// TIA Portal V16 export
// export: Created 2021-07-03T21:22:43.1063797Z, ExportSetting WithDefaults, DisplayName Totally Integrated Automation Portal, DisplayVersion V16, DisplayName TIA Portal Version Control Interface, DisplayVersion V16, DisplayName TIA Portal Openness, DisplayVersion V16, DisplayName STEP 7 Professional, DisplayVersion V16, DisplayName STEP 7 Safety, DisplayVersion V16, DisplayName WinCC Professional, DisplayVersion V16
TYPE "118MK2_UPIF_Status"
// stored: IsFailsafeCompliant false
   STRUCT
      PLANT_TAG_NAME { ExternalAccessible := 'False'; ExternalVisible := 'False'; ExternalWritable := 'False'} : Array[0..15] of Byte;   // Current plant tag name of the sorting module, 16 character string
      UP_MACHINE_NAME { ExternalAccessible := 'False'; ExternalVisible := 'False'; ExternalWritable := 'False'} : Array[0..15] of Byte;   // Current manufacturer name of the sorting module – read from the cRIO Controller configuration, 16-character string
      COMMAND_ACK_S { ExternalAccessible := 'False'; ExternalVisible := 'False'; ExternalWritable := 'False'} : Byte;   // Returns the (same) command value as an acknowledgement that the Real-time system has received the command.
      COMMAND_IN_PROG_S { ExternalAccessible := 'False'; ExternalVisible := 'False'; ExternalWritable := 'False'} : Byte;   // Counts up as progress indicator – resets on completion
      INVALID_COMMAND_S { ExternalAccessible := 'False'; ExternalVisible := 'False'; ExternalWritable := 'False'} : Bool;   // ‘1’ when an invalid command – cleared on next valid command.
      PARAM_OUT_OF_RANGE_S { ExternalAccessible := 'False'; ExternalVisible := 'False'; ExternalWritable := 'False'} : Bool;   // ‘1’ when any requested parameter value is out of range.
      USER_ADDED_S { ExternalAccessible := 'False'; ExternalVisible := 'False'; ExternalWritable := 'False'} : Bool;   // ‘1’ when a requested new user name was successfully added to the security lookup table.
      PASSWORD_CHANGED_S { ExternalAccessible := 'False'; ExternalVisible := 'False'; ExternalWritable := 'False'} : Bool;   // ‘1’ when a requested password change was successful.
      USER_DELETED_S { ExternalAccessible := 'False'; ExternalVisible := 'False'; ExternalWritable := 'False'} : Bool;   // ‘1’ temporarily when a requested user delete was successful
      LOGON_ATTEMPT_FAILED_S { ExternalAccessible := 'False'; ExternalVisible := 'False'; ExternalWritable := 'False'} : Bool;   // ‘1’ temporarily when a logon attempt failed.
      NO_XRAY_DOOR_OPEN_S { ExternalAccessible := 'False'; ExternalVisible := 'False'; ExternalWritable := 'False'} : Bool;   // ‘1’ temporarily when no X-rays possible because doors are open.
      NO_OPP_INCOM_AIR_LOW_S { ExternalAccessible := 'False'; ExternalVisible := 'False'; ExternalWritable := 'False'} : Bool;   // ‘1’ temporarily when no operation possible due to low air pressure.
      GLOBAL_ALARM_S { ExternalAccessible := 'False'; ExternalVisible := 'False'; ExternalWritable := 'False'} : Bool;   // ‘1’ when any alarm is present. Cleared when all alarms are reset.
      OTI_COMMS_FAULT_S { ExternalAccessible := 'False'; ExternalVisible := 'False'; ExternalWritable := 'False'} : Bool;   // ‘1’ when comms fault between OTI and cRIO.
      LOCAL_REMOTE_S { ExternalAccessible := 'False'; ExternalVisible := 'False'; ExternalWritable := 'False'} : Bool;   // ‘1’ when machine is in Remote mode
      MAINTENANCE_MODE_S { ExternalAccessible := 'False'; ExternalVisible := 'False'; ExternalWritable := 'False'} : Bool;   // ‘1’ when in Maintenance Mode
      INCOM_AIR_PRESS_LO_S { ExternalAccessible := 'False'; ExternalVisible := 'False'; ExternalWritable := 'False'} : Bool;   // ‘1’ when incoming air pressure less than low setpoint i.e. 4.5 bar.
      INCOM_AIR_PRESS_LOLO_S { ExternalAccessible := 'False'; ExternalVisible := 'False'; ExternalWritable := 'False'} : Bool;   // ‘1’ when incoming air pressure less than low low setpoint i.e. 4.0 bar.
      PROC_WATERFLOW_HIGH_S { ExternalAccessible := 'False'; ExternalVisible := 'False'; ExternalWritable := 'False'} : Bool;   // ‘1’ when flow rate greater than flow set-point plus allowed deviation.
      PROC_WATERFLOW_LOW_S { ExternalAccessible := 'False'; ExternalVisible := 'False'; ExternalWritable := 'False'} : Bool;   // ‘1’ when flow rate less than flow set-point minus allowed deviation.
      FEEDER_RUNNING_S { ExternalAccessible := 'False'; ExternalVisible := 'False'; ExternalWritable := 'False'} : Bool;   // ‘1’ when feeder is running.
      REMOTE_DNSTRM_INTLK_S { ExternalAccessible := 'False'; ExternalVisible := 'False'; ExternalWritable := 'False'} : Bool;   // ‘1’ when downstream interlock healthy from PLC.
      HOLD_STATE_S { ExternalAccessible := 'False'; ExternalVisible := 'False'; ExternalWritable := 'False'} : Bool;   // ‘1’ when feeder is prevented from running in “Processing” due to process interlock, low air pressure etc.
      WAIT_STATE_S { ExternalAccessible := 'False'; ExternalVisible := 'False'; ExternalWritable := 'False'} : Bool;   // ‘1’ when in “Processing” state.
      PURGED_STATE_S { ExternalAccessible := 'False'; ExternalVisible := 'False'; ExternalWritable := 'False'} : Bool;   // ‘1’ when a purge cycle is successfully completed. Cleared when feeder is next started.
      EJECTION_RATE_WARN_S { ExternalAccessible := 'False'; ExternalVisible := 'False'; ExternalWritable := 'False'} : Bool;   // ‘1’ when ejection rate exceeds warning level.
      EJECTION_RATE_ALARM_S { ExternalAccessible := 'False'; ExternalVisible := 'False'; ExternalWritable := 'False'} : Bool;   // ‘1’ when ejection rate exceeded ejection rate alarm level.
      MACH_ESTOP_ACTIVE_S { ExternalAccessible := 'False'; ExternalVisible := 'False'; ExternalWritable := 'False'} : Bool;   // ‘1’ when E-stop active.
      XRAY_COOLW_TEMP_FAULT_S { ExternalAccessible := 'False'; ExternalVisible := 'False'; ExternalWritable := 'False'} : Bool;   // ‘1’ when X-ray cooling water temperature to high or too low fault detected.
      XRAY_COOLW_FLOW_FAULT_S { ExternalAccessible := 'False'; ExternalVisible := 'False'; ExternalWritable := 'False'} : Bool;   // ‘1’ when cooling water flow low fault detected.
      PROC_WATER_FLOW_S { ExternalAccessible := 'False'; ExternalVisible := 'False'; ExternalWritable := 'False'} : Bool;   // ‘1’ when process water flow too high or too low fault detected. (Wet machine only)
      FRONT_SIDE_PROC_DOOR_S { ExternalAccessible := 'False'; ExternalVisible := 'False'; ExternalWritable := 'False'} : Bool;   // ‘1’ when front side door open.
      BACK_SIDE_PROC_DOOR_S { ExternalAccessible := 'False'; ExternalVisible := 'False'; ExternalWritable := 'False'} : Bool;   // ‘1’ when back side door open.
      FEEDER_DOOR_S { ExternalAccessible := 'False'; ExternalVisible := 'False'; ExternalWritable := 'False'} : Bool;   // ‘1’ when feeder door open.
      HOOD_S { ExternalAccessible := 'False'; ExternalVisible := 'False'; ExternalWritable := 'False'} : Bool;   // ‘1’ when hood open.
      CONC_TRACER_DOOR_S { ExternalAccessible := 'False'; ExternalVisible := 'False'; ExternalWritable := 'False'} : Bool;   // ‘1’ when concentrate tracer door open.
      TAILINGS_TRACER_DOOR_S { ExternalAccessible := 'False'; ExternalVisible := 'False'; ExternalWritable := 'False'} : Bool;   // ‘1’ when tailings tracer door open.
      CONC_TRACER_TRAY_S { ExternalAccessible := 'False'; ExternalVisible := 'False'; ExternalWritable := 'False'} : Bool;   // ‘1’ when concentrate tracer tray in position.
      TAILINGS_TRACER_TRAY_S { ExternalAccessible := 'False'; ExternalVisible := 'False'; ExternalWritable := 'False'} : Bool;   // ‘1’ when tailings tracer tray in position.
      PLANT_INLET_CHUTE_S { ExternalAccessible := 'False'; ExternalVisible := 'False'; ExternalWritable := 'False'} : Bool;   // ‘1’ when plant inlet not in position.
      INSPECTION_COVER_S { ExternalAccessible := 'False'; ExternalVisible := 'False'; ExternalWritable := 'False'} : Bool;   // ‘1’ when inspection cover not in position.
      PLANT_CONC_CHUTE_S { ExternalAccessible := 'False'; ExternalVisible := 'False'; ExternalWritable := 'False'} : Bool;   // ‘1’ when plant concentrate chute not in position.
      PLANT_TAILINGS_CHUTE_S { ExternalAccessible := 'False'; ExternalVisible := 'False'; ExternalWritable := 'False'} : Bool;   // ‘1’ when plant tailings chute not in position.
      INTERN_CONC_CHUTE_S { ExternalAccessible := 'False'; ExternalVisible := 'False'; ExternalWritable := 'False'} : Bool;   // ‘1’ when internal concentrate chute not in position.
      INTERN_TAILINGS_CHUTE_S { ExternalAccessible := 'False'; ExternalVisible := 'False'; ExternalWritable := 'False'} : Bool;   // ‘1’ when internal tailings chute not in position.
      DUSTEXTRACT_FLOW_FLT_S { ExternalAccessible := 'False'; ExternalVisible := 'False'; ExternalWritable := 'False'} : Bool;   // ‘1’ when dust extractor flow fault detected (Dry machine only)
      SURGE_ARRESTOR_FLT_S { ExternalAccessible := 'False'; ExternalVisible := 'False'; ExternalWritable := 'False'} : Bool;   // ‘1’ when one or more surge arrestors on the electrical panel is faulty.
      DXM_XRAY_GEN_COMM_FLT_S { ExternalAccessible := 'False'; ExternalVisible := 'False'; ExternalWritable := 'False'} : Bool;   // ‘1’ when no comms between cRIO and Spellman DXM X-ray generator.
      DXM_HV_ENABLED_S { ExternalAccessible := 'False'; ExternalVisible := 'False'; ExternalWritable := 'False'} : Bool;   // ‘1’ when X-rays ON.
      DXM_INTERLOCK_CLOSED_S { ExternalAccessible := 'False'; ExternalVisible := 'False'; ExternalWritable := 'False'} : Bool;   // ‘1’ when interlock on X-ray generator is healthy.
      DXM_PS_FLT_S { ExternalAccessible := 'False'; ExternalVisible := 'False'; ExternalWritable := 'False'} : Bool;   // ‘1’ when X-ray generator power supply fault detected.
      STATUS_BYTE6_SPARE7 { ExternalAccessible := 'False'; ExternalVisible := 'False'; ExternalWritable := 'False'} : Bool;   // Status Byte-6 Spare
      STATUS_BYTE7_SPARE0 { ExternalAccessible := 'False'; ExternalVisible := 'False'; ExternalWritable := 'False'} : Bool;   // Status Byte-7 Spare
      STATUS_BYTE7_SPARE1 { ExternalAccessible := 'False'; ExternalVisible := 'False'; ExternalWritable := 'False'} : Bool;   // Status Byte-7 Spare
      STATUS_BYTE7_SPARE2 { ExternalAccessible := 'False'; ExternalVisible := 'False'; ExternalWritable := 'False'} : Bool;   // Status Byte-7 Spare
      STATUS_BYTE7_SPARE3 { ExternalAccessible := 'False'; ExternalVisible := 'False'; ExternalWritable := 'False'} : Bool;   // Status Byte-7 Spare
      STATUS_BYTE7_SPARE4 { ExternalAccessible := 'False'; ExternalVisible := 'False'; ExternalWritable := 'False'} : Bool;   // Status Byte-7 Spare
      STATUS_BYTE7_SPARE5 { ExternalAccessible := 'False'; ExternalVisible := 'False'; ExternalWritable := 'False'} : Bool;   // Status Byte-7 Spare
      STATUS_BYTE7_SPARE6 { ExternalAccessible := 'False'; ExternalVisible := 'False'; ExternalWritable := 'False'} : Bool;   // Status Byte-7 Spare
      STATUS_BYTE7_SPARE7 { ExternalAccessible := 'False'; ExternalVisible := 'False'; ExternalWritable := 'False'} : Bool;   // Status Byte-7 Spare
      STATUS_BYTE8_SPARE0 { ExternalAccessible := 'False'; ExternalVisible := 'False'; ExternalWritable := 'False'} : Bool;   // Status Byte-8 Spare
      STATUS_BYTE8_SPARE1 { ExternalAccessible := 'False'; ExternalVisible := 'False'; ExternalWritable := 'False'} : Bool;   // Status Byte-8 Spare
      STATUS_BYTE8_SPARE2 { ExternalAccessible := 'False'; ExternalVisible := 'False'; ExternalWritable := 'False'} : Bool;   // Status Byte-8 Spare
      STATUS_BYTE8_SPARE3 { ExternalAccessible := 'False'; ExternalVisible := 'False'; ExternalWritable := 'False'} : Bool;   // Status Byte-8 Spare
      STATUS_BYTE8_SPARE4 { ExternalAccessible := 'False'; ExternalVisible := 'False'; ExternalWritable := 'False'} : Bool;   // Status Byte-8 Spare
      STATUS_BYTE8_SPARE5 { ExternalAccessible := 'False'; ExternalVisible := 'False'; ExternalWritable := 'False'} : Bool;   // Status Byte-8 Spare
      STATUS_BYTE8_SPARE6 { ExternalAccessible := 'False'; ExternalVisible := 'False'; ExternalWritable := 'False'} : Bool;   // Status Byte-8 Spare
      STATUS_BYTE8_SPARE7 { ExternalAccessible := 'False'; ExternalVisible := 'False'; ExternalWritable := 'False'} : Bool;   // Status Byte-8 Spare
      STATUS_BYTE9_SPARE0 { ExternalAccessible := 'False'; ExternalVisible := 'False'; ExternalWritable := 'False'} : Bool;   // Status Byte-9 Spare
      STATUS_BYTE9_SPARE1 { ExternalAccessible := 'False'; ExternalVisible := 'False'; ExternalWritable := 'False'} : Bool;   // Status Byte-9 Spare
      STATUS_BYTE9_SPARE2 { ExternalAccessible := 'False'; ExternalVisible := 'False'; ExternalWritable := 'False'} : Bool;   // Status Byte-9 Spare
      STATUS_BYTE9_SPARE3 { ExternalAccessible := 'False'; ExternalVisible := 'False'; ExternalWritable := 'False'} : Bool;   // Status Byte-9 Spare
      STATUS_BYTE9_SPARE4 { ExternalAccessible := 'False'; ExternalVisible := 'False'; ExternalWritable := 'False'} : Bool;   // Status Byte-9 Spare
      STATUS_BYTE9_SPARE5 { ExternalAccessible := 'False'; ExternalVisible := 'False'; ExternalWritable := 'False'} : Bool;   // Status Byte-9 Spare
      STATUS_BYTE9_SPARE6 { ExternalAccessible := 'False'; ExternalVisible := 'False'; ExternalWritable := 'False'} : Bool;   // Status Byte-9 Spare
      STATUS_BYTE9_SPARE7 { ExternalAccessible := 'False'; ExternalVisible := 'False'; ExternalWritable := 'False'} : Bool;   // Status Byte-9 Spare
      STATUS_BYTE10_SPARE0 { ExternalAccessible := 'False'; ExternalVisible := 'False'; ExternalWritable := 'False'} : Bool;   // Status Byte-10 Spare
      STATUS_BYTE10_SPARE1 { ExternalAccessible := 'False'; ExternalVisible := 'False'; ExternalWritable := 'False'} : Bool;   // Status Byte-10 Spare
      STATUS_BYTE10_SPARE2 { ExternalAccessible := 'False'; ExternalVisible := 'False'; ExternalWritable := 'False'} : Bool;   // Status Byte-10 Spare
      STATUS_BYTE10_SPARE3 { ExternalAccessible := 'False'; ExternalVisible := 'False'; ExternalWritable := 'False'} : Bool;   // Status Byte-10 Spare
      STATUS_BYTE10_SPARE4 { ExternalAccessible := 'False'; ExternalVisible := 'False'; ExternalWritable := 'False'} : Bool;   // Status Byte-10 Spare
      STATUS_BYTE10_SPARE5 { ExternalAccessible := 'False'; ExternalVisible := 'False'; ExternalWritable := 'False'} : Bool;   // Status Byte-10 Spare
      STATUS_BYTE10_SPARE6 { ExternalAccessible := 'False'; ExternalVisible := 'False'; ExternalWritable := 'False'} : Bool;   // Status Byte-10 Spare
      STATUS_BYTE10_SPARE7 { ExternalAccessible := 'False'; ExternalVisible := 'False'; ExternalWritable := 'False'} : Bool;   // Status Byte-10 Spare
      MACHINE_STATE_S { ExternalAccessible := 'False'; ExternalVisible := 'False'; ExternalWritable := 'False'} : Byte;   // 0-Initializing, 1-Ready, 2-Purging, 3-Display, 4-Calibrating, 5-Checker Cycle, 6-Processing Ready, 7-Processing, 8-Transition, 9-Alarm.
      DXM_COMMS_FLT_A { ExternalAccessible := 'False'; ExternalVisible := 'False'; ExternalWritable := 'False'} : Bool;   // ALARM: DXM Comms fault
      DXM_XRAY_STATE_A { ExternalAccessible := 'False'; ExternalVisible := 'False'; ExternalWritable := 'False'} : Bool;   // ALARM: DXM X-ray state alarm
      DXM_INTERLOCK_FLT_A { ExternalAccessible := 'False'; ExternalVisible := 'False'; ExternalWritable := 'False'} : Bool;   // ALARM: DXM Interlock fault
      DXM_PSU_FAULT_A { ExternalAccessible := 'False'; ExternalVisible := 'False'; ExternalWritable := 'False'} : Bool;   // ALARM: DXM Power supply fault
      DXM_NOTIN_REM_MODE_A { ExternalAccessible := 'False'; ExternalVisible := 'False'; ExternalWritable := 'False'} : Bool;   // ALARM: DXM Not in remote mode fault
      DXM_ARC_FLT_A { ExternalAccessible := 'False'; ExternalVisible := 'False'; ExternalWritable := 'False'} : Bool;   // ALARM: DXM Arc fault
      DXM_OVER_TEMP_FLT_A { ExternalAccessible := 'False'; ExternalVisible := 'False'; ExternalWritable := 'False'} : Bool;   // ALARM: DXM Over temperature fault
      DXM_OVER_VOLT_FLT_A { ExternalAccessible := 'False'; ExternalVisible := 'False'; ExternalWritable := 'False'} : Bool;   // ALARM: DXM Over voltage fault
      DXM_UNDER_VOLT_FLT_A { ExternalAccessible := 'False'; ExternalVisible := 'False'; ExternalWritable := 'False'} : Bool;   // ALARM: DXM Under voltage fault
      DXM_OVER_CURRENT_FLT_A { ExternalAccessible := 'False'; ExternalVisible := 'False'; ExternalWritable := 'False'} : Bool;   // ALARM: DXM Over current fault
      DXM_UNDER_CURRENT_FLT_A { ExternalAccessible := 'False'; ExternalVisible := 'False'; ExternalWritable := 'False'} : Bool;   // ALARM: DXM Under current fault
      DXM_MODEL_NUMB_FLT_A { ExternalAccessible := 'False'; ExternalVisible := 'False'; ExternalWritable := 'False'} : Bool;   // ALARM: DXM Model number fault
      ASI_COMMS_FAULT_A { ExternalAccessible := 'False'; ExternalVisible := 'False'; ExternalWritable := 'False'} : Bool;   // ALARM: ASI Comms fault
      ASI_MISSING_SLAVE_FLT_A { ExternalAccessible := 'False'; ExternalVisible := 'False'; ExternalWritable := 'False'} : Bool;   // ALARM: ASI Missing slave fault
      ASI_DUPL_SLAVE_FLT_A { ExternalAccessible := 'False'; ExternalVisible := 'False'; ExternalWritable := 'False'} : Bool;   // ALARM: ASI Duplicate slave fault
      ASI_UNAUTH_SLAVE_FLT_A { ExternalAccessible := 'False'; ExternalVisible := 'False'; ExternalWritable := 'False'} : Bool;   // ALARM: ASI Unauthorised slave fault
      ASIBUS_VOLT_LO_A { ExternalAccessible := 'False'; ExternalVisible := 'False'; ExternalWritable := 'False'} : Bool;   // ALARM: ASI Bus voltage less than 28Vdc
      ASI_PERIP_FLT_A { ExternalAccessible := 'False'; ExternalVisible := 'False'; ExternalWritable := 'False'} : Bool;   // ALARM: ASI Peripheral fault
      ASIBUS_VOLTS_EARTH_FLT_A { ExternalAccessible := 'False'; ExternalVisible := 'False'; ExternalWritable := 'False'} : Bool;   // ALARM: ASI Bus voltage earth fault
      CRIO_MPLC_COMMS_FAIL_A { ExternalAccessible := 'False'; ExternalVisible := 'False'; ExternalWritable := 'False'} : Bool;   // ALARM: cRIO - Machine PLC Comms failure
      CRIO_CHAS_TEMP_TOOHIGH_A { ExternalAccessible := 'False'; ExternalVisible := 'False'; ExternalWritable := 'False'} : Bool;   // ALARM: cRIO chassis temperature too high
      XRAYGEN_COMP_TEMPHIGH_A { ExternalAccessible := 'False'; ExternalVisible := 'False'; ExternalWritable := 'False'} : Bool;   // ALARM: X-ray generator compartment temperature high
      FPGA_HEARTBEAT_ERR_A { ExternalAccessible := 'False'; ExternalVisible := 'False'; ExternalWritable := 'False'} : Bool;   // ALARM: FPGA heartbeat error
      FPGA_MODE_ERR_A { ExternalAccessible := 'False'; ExternalVisible := 'False'; ExternalWritable := 'False'} : Bool;   // ALARM: FPGA mode error
      EJECT_FIRE_RATE_A { ExternalAccessible := 'False'; ExternalVisible := 'False'; ExternalWritable := 'False'} : Bool;   // ALARM: Ejector fire rate alarm
      FEED_RATE_A { ExternalAccessible := 'False'; ExternalVisible := 'False'; ExternalWritable := 'False'} : Bool;   // ALARM: Feed rate alarm
      COOLWATER_TEMP_HIGH_A { ExternalAccessible := 'False'; ExternalVisible := 'False'; ExternalWritable := 'False'} : Bool;   // ALARM: Cooling water temperature high
      COOLWATER_TEMP_LOW_A { ExternalAccessible := 'False'; ExternalVisible := 'False'; ExternalWritable := 'False'} : Bool;   // ALARM: Cooling water temperature low
      COOLWATER_FLOW_LO_A { ExternalAccessible := 'False'; ExternalVisible := 'False'; ExternalWritable := 'False'} : Bool;   // ALARM: Cooling water flow low
      PROCWATER_FLOW_LO_ERR_A { ExternalAccessible := 'False'; ExternalVisible := 'False'; ExternalWritable := 'False'} : Bool;   // ALARM: Process water flow low error
      PROCWATER_FLOW_HI_ERR_A { ExternalAccessible := 'False'; ExternalVisible := 'False'; ExternalWritable := 'False'} : Bool;   // ALARM: Process water flow high error
      INCOM_AIRPRESS_LO_A { ExternalAccessible := 'False'; ExternalVisible := 'False'; ExternalWritable := 'False'} : Bool;   // ALARM: Incoming air pressure low
      CALJIG_NOT_EXTEND_FLT_A { ExternalAccessible := 'False'; ExternalVisible := 'False'; ExternalWritable := 'False'} : Bool;   // ALARM: Calibration jig not extending fault
      CALJIG_NOT_RETRACT_FLT_A { ExternalAccessible := 'False'; ExternalVisible := 'False'; ExternalWritable := 'False'} : Bool;   // ALARM: Calibration jig not retracting fault
      CALJIGDR_NOT_OPEN_FLT_A { ExternalAccessible := 'False'; ExternalVisible := 'False'; ExternalWritable := 'False'} : Bool;   // ALARM: Calibration jig door not opening fault
      CALJIGDR_NOT_CLOS_FLT_A { ExternalAccessible := 'False'; ExternalVisible := 'False'; ExternalWritable := 'False'} : Bool;   // ALARM: Calibration jig door not closing fault
      CALIB_DEV_ERR_A { ExternalAccessible := 'False'; ExternalVisible := 'False'; ExternalWritable := 'False'} : Bool;   // ALARM: Calibration deviation error
      CHANNEL_DATA_ZERO_A { ExternalAccessible := 'False'; ExternalVisible := 'False'; ExternalWritable := 'False'} : Bool;   // ALARM: Channel data zero
      EJECTOR_ERRORS_A { ExternalAccessible := 'False'; ExternalVisible := 'False'; ExternalWritable := 'False'} : Bool;   // ALARM: Ejector error(s)
      FRONT_SIDE_DR_OPN_A { ExternalAccessible := 'False'; ExternalVisible := 'False'; ExternalWritable := 'False'} : Bool;   // ALARM: Front side door open
      BACK_SIDE_DR_OPN_A { ExternalAccessible := 'False'; ExternalVisible := 'False'; ExternalWritable := 'False'} : Bool;   // ALARM: Back side door open
      FEEDER_DOOR_OPN_A { ExternalAccessible := 'False'; ExternalVisible := 'False'; ExternalWritable := 'False'} : Bool;   // ALARM: Feeder door open
      CONC_TRACERDR_OPN_A { ExternalAccessible := 'False'; ExternalVisible := 'False'; ExternalWritable := 'False'} : Bool;   // ALARM: Concentrate tracer door open
      TAILS_TRACERDR_OPN_A { ExternalAccessible := 'False'; ExternalVisible := 'False'; ExternalWritable := 'False'} : Bool;   // ALARM: Tailings tracer door open
      HOOD_OPEN_A { ExternalAccessible := 'False'; ExternalVisible := 'False'; ExternalWritable := 'False'} : Bool;   // ALARM: Hood open
      P_INLET_CHTE_NOTINPOS_A { ExternalAccessible := 'False'; ExternalVisible := 'False'; ExternalWritable := 'False'} : Bool;   // ALARM: Plant inlet chute not in position
      INSPEC_COVER_OPN_A { ExternalAccessible := 'False'; ExternalVisible := 'False'; ExternalWritable := 'False'} : Bool;   // ALARM: Inspection cover open
      P_CONC_CHTE_NOTINPOS_A { ExternalAccessible := 'False'; ExternalVisible := 'False'; ExternalWritable := 'False'} : Bool;   // ALARM: Plant concentrate chute not in position
      P_TAILS_CHTE_NOTINPOS_A { ExternalAccessible := 'False'; ExternalVisible := 'False'; ExternalWritable := 'False'} : Bool;   // ALARM: Plant tailings chute not in position
      INTCONC_CHTE_NOTINPOS_A { ExternalAccessible := 'False'; ExternalVisible := 'False'; ExternalWritable := 'False'} : Bool;   // ALARM: Internal concentrate chute not in position
      INTTAILS_CHTE_NOTINPOS_A { ExternalAccessible := 'False'; ExternalVisible := 'False'; ExternalWritable := 'False'} : Bool;   // ALARM: Internal tailings chute not in position
      DUST_EXTRACT_FLOW_FLT_A { ExternalAccessible := 'False'; ExternalVisible := 'False'; ExternalWritable := 'False'} : Bool;   // ALARM: Dust extractor flow fault
      GATE_POSITION_FLT_A { ExternalAccessible := 'False'; ExternalVisible := 'False'; ExternalWritable := 'False'} : Bool;   // ALARM: Gate position fault
      MACH_ESTOP_PRESSED_A { ExternalAccessible := 'False'; ExternalVisible := 'False'; ExternalWritable := 'False'} : Bool;   // ALARM: Machine E-Stop button pressed
      SURGE_ARREST_FLT_A { ExternalAccessible := 'False'; ExternalVisible := 'False'; ExternalWritable := 'False'} : Bool;   // ALARM: Surge arrestor fault
      ASI_SAFETY_BRIDGE_MISS_A { ExternalAccessible := 'False'; ExternalVisible := 'False'; ExternalWritable := 'False'} : Bool;   // ALARM: ASI Safety bridging plug missing
      ASI_ESTOP_CONT_FB_FLT_A { ExternalAccessible := 'False'; ExternalVisible := 'False'; ExternalWritable := 'False'} : Bool;   // ALARM: ASI E-stop contactor feedback fault
      XRAY_CONT_FB_FLT_A { ExternalAccessible := 'False'; ExternalVisible := 'False'; ExternalWritable := 'False'} : Bool;   // ALARM: X-ray contactors feedback fault
      TRACERTRAY_INPOS_REM_A { ExternalAccessible := 'False'; ExternalVisible := 'False'; ExternalWritable := 'False'} : Bool;   // ALARM: Tracer tray/s in position in remote mode
      CALIBJIG_COVR_NOTINPOS_A { ExternalAccessible := 'False'; ExternalVisible := 'False'; ExternalWritable := 'False'} : Bool;   // ALARM: Calibration jig cover not in position
      ASI_ESTOP_CONT_FAIL_A { ExternalAccessible := 'False'; ExternalVisible := 'False'; ExternalWritable := 'False'} : Bool;   // ALARM: ASI E-stop contactor failure
      ASI_PROJSLV_FLT_A { ExternalAccessible := 'False'; ExternalVisible := 'False'; ExternalWritable := 'False'} : Bool;   // ALARM: ASI Projected slaves’ fault
      ASI_PARAM_OUTP_FLT_A { ExternalAccessible := 'False'; ExternalVisible := 'False'; ExternalWritable := 'False'} : Bool;   // ALARM: ASI Parameter output fault
      ASISAFE_DEV_CODE_FLT_A { ExternalAccessible := 'False'; ExternalVisible := 'False'; ExternalWritable := 'False'} : Bool;   // ALARM: ASI Safety device code fault
      "ASISAFE_PLC COMM_FLT_A" { ExternalAccessible := 'False'; ExternalVisible := 'False'; ExternalWritable := 'False'} : Bool;   // ALARM: ASI Safety PLC comms alarm
      ASIBUS_VOLT_ASSYM_A { ExternalAccessible := 'False'; ExternalVisible := 'False'; ExternalWritable := 'False'} : Bool;   // ALARM: ASi Bus voltage asymmetrical
      FILMW_EMPTY_FLT_A { ExternalAccessible := 'False'; ExternalVisible := 'False'; ExternalWritable := 'False'} : Bool;   // ALARM: Film Winder empty fault
      FILMW_TORN_FLT_A { ExternalAccessible := 'False'; ExternalVisible := 'False'; ExternalWritable := 'False'} : Bool;   // ALARM: Film Winder torn fault
      FILMW_NOTROT_FLT_A { ExternalAccessible := 'False'; ExternalVisible := 'False'; ExternalWritable := 'False'} : Bool;   // ALARM: Film Winder not rotating fault
      FILMW_TIMOUT_A { ExternalAccessible := 'False'; ExternalVisible := 'False'; ExternalWritable := 'False'} : Bool;   // ALARM: Film Winder timeout
      FILMW_COM_TIMOUT_FLT_A { ExternalAccessible := 'False'; ExternalVisible := 'False'; ExternalWritable := 'False'} : Bool;   // ALARM: Film Winder comms timeout fault
      FILMWIND_MOT_A { ExternalAccessible := 'False'; ExternalVisible := 'False'; ExternalWritable := 'False'} : Bool;   // ALARM: Film Winder motor alarm
      FILMWIND_UNKN_FLT_A { ExternalAccessible := 'False'; ExternalVisible := 'False'; ExternalWritable := 'False'} : Bool;   // ALARM: Film Winder unknown fault
      DXM_KV_DEV_FLT_A { ExternalAccessible := 'False'; ExternalVisible := 'False'; ExternalWritable := 'False'} : Bool;   // ALARM: DXM KV deviation fault
      DXM_MA_DEV_FLT_A { ExternalAccessible := 'False'; ExternalVisible := 'False'; ExternalWritable := 'False'} : Bool;   // ALARM: DXM mA deviation fault
      ASI_SOFTW_NUM_FLT_A { ExternalAccessible := 'False'; ExternalVisible := 'False'; ExternalWritable := 'False'} : Bool;   // ALARM: AS-i Software Number fault
      ALARM_BYTE10_SPARE4 { ExternalAccessible := 'False'; ExternalVisible := 'False'; ExternalWritable := 'False'} : Bool;   // Alarm Byte-10 Spare
      ALARM_BYTE10_SPARE5 { ExternalAccessible := 'False'; ExternalVisible := 'False'; ExternalWritable := 'False'} : Bool;   // Alarm Byte-10 Spare
      ALARM_BYTE10_SPARE6 { ExternalAccessible := 'False'; ExternalVisible := 'False'; ExternalWritable := 'False'} : Bool;   // Alarm Byte-10 Spare
      ALARM_BYTE10_SPARE7 { ExternalAccessible := 'False'; ExternalVisible := 'False'; ExternalWritable := 'False'} : Bool;   // Alarm Byte-10 Spare
      ALARM_BYTE11_SPARE0 { ExternalAccessible := 'False'; ExternalVisible := 'False'; ExternalWritable := 'False'} : Bool;   // Alarm Byte-11 Spare
      ALARM_BYTE11_SPARE1 { ExternalAccessible := 'False'; ExternalVisible := 'False'; ExternalWritable := 'False'} : Bool;   // Alarm Byte-11 Spare
      ALARM_BYTE11_SPARE2 { ExternalAccessible := 'False'; ExternalVisible := 'False'; ExternalWritable := 'False'} : Bool;   // Alarm Byte-11 Spare
      ALARM_BYTE11_SPARE3 { ExternalAccessible := 'False'; ExternalVisible := 'False'; ExternalWritable := 'False'} : Bool;   // Alarm Byte-11 Spare
      ALARM_BYTE11_SPARE4 { ExternalAccessible := 'False'; ExternalVisible := 'False'; ExternalWritable := 'False'} : Bool;   // Alarm Byte-11 Spare
      ALARM_BYTE11_SPARE5 { ExternalAccessible := 'False'; ExternalVisible := 'False'; ExternalWritable := 'False'} : Bool;   // Alarm Byte-11 Spare
      ALARM_BYTE11_SPARE6 { ExternalAccessible := 'False'; ExternalVisible := 'False'; ExternalWritable := 'False'} : Bool;   // Alarm Byte-11 Spare
      ALARM_BYTE11_SPARE7 { ExternalAccessible := 'False'; ExternalVisible := 'False'; ExternalWritable := 'False'} : Bool;   // Alarm Byte-11 Spare
      RECPAR_EJ_DELTIME_ACT { ExternalAccessible := 'False'; ExternalVisible := 'False'; ExternalWritable := 'False'} : Byte;   // Recipe Parameter: Ejector Delay Time Actual, (0 to 50ms)
      RECPAR_EJ_ONTIME_ACT { ExternalAccessible := 'False'; ExternalVisible := 'False'; ExternalWritable := 'False'} : Byte;   // Recipe Parameter: Ejection On Time Actual, (1 to 50ms)
      RECPAR_BLINT_TH_ACT { ExternalAccessible := 'False'; ExternalVisible := 'False'; ExternalWritable := 'False'} : Word;   // Recipe Parameter: Algorithm Blue Intensity Threshold Actual, (60 to 10000mV)
      RECPAR_BLRD_OFF_ACT { ExternalAccessible := 'False'; ExternalVisible := 'False'; ExternalWritable := 'False'} : Word;   // Recipe Parameter: Algorithm Blue-Red Discrimination Offset Actual, (0 to 10000)
      RECPAR_BLRD_RAT_ACT { ExternalAccessible := 'False'; ExternalVisible := 'False'; ExternalWritable := 'False'} : Word;   // Recipe Parameter: Algorithm Blue-Red Discrimination Ratio Actual, (1 to 1000 equiv. 0.01 to 10.00)
      RECPAR_VIBFEED_SP_ACT { ExternalAccessible := 'False'; ExternalVisible := 'False'; ExternalWritable := 'False'} : Byte;   // Recipe Parameter: Vibratory Feeder Setpoint Actual, (0 to 100%)
      RECPAR_AUTFEEDC_ACT { ExternalAccessible := 'False'; ExternalVisible := 'False'; ExternalWritable := 'False'} : Bool;   // Recipe Parameter: Automatic Feeder Control Actual, OFF(0) – No closed loop control, ON(1) – Closed loop control
      RECPAR_RESERVED1 { ExternalAccessible := 'False'; ExternalVisible := 'False'; ExternalWritable := 'False'} : Bool;   // Recipe Parameter: Reserved - Do Not Use
      RECPAR_RESERVED2 { ExternalAccessible := 'False'; ExternalVisible := 'False'; ExternalWritable := 'False'} : Bool;   // Recipe Parameter: Reserved - Do Not Use
      RECPAR_RESERVED3 { ExternalAccessible := 'False'; ExternalVisible := 'False'; ExternalWritable := 'False'} : Bool;   // Recipe Parameter: Reserved - Do Not Use
      RECPAR_RESERVED4 { ExternalAccessible := 'False'; ExternalVisible := 'False'; ExternalWritable := 'False'} : Bool;   // Recipe Parameter: Reserved - Do Not Use
      RECPAR_RESERVED5 { ExternalAccessible := 'False'; ExternalVisible := 'False'; ExternalWritable := 'False'} : Bool;   // Recipe Parameter: Reserved - Do Not Use
      RECPAR_RESERVED6 { ExternalAccessible := 'False'; ExternalVisible := 'False'; ExternalWritable := 'False'} : Bool;   // Recipe Parameter: Reserved - Do Not Use
      RECPAR_RESERVED7 { ExternalAccessible := 'False'; ExternalVisible := 'False'; ExternalWritable := 'False'} : Bool;   // Recipe Parameter: Reserved - Do Not Use
      RECPAR_GATEPOS_ACT { ExternalAccessible := 'False'; ExternalVisible := 'False'; ExternalWritable := 'False'} : Byte;   // Recipe Parameter: Gate Position Actual - ‘0’ - No auto gate, ‘1’ - Gate in position 1(-2 +1mm), ‘2’ – Gate in position 2(-4+2mm), ‘3’ – Gate in position 3(-8+4mm), ‘4’ – Gate in position 4(-16+8mm), ‘5’ – Gate in position 5(-32+16mm)
      SPARE0 { ExternalAccessible := 'False'; ExternalVisible := 'False'; ExternalWritable := 'False'} : Byte;   // Spare
      SPARE1 { ExternalAccessible := 'False'; ExternalVisible := 'False'; ExternalWritable := 'False'} : DWord;   // Spare
      SPARE2 { ExternalAccessible := 'False'; ExternalVisible := 'False'; ExternalWritable := 'False'} : DWord;   // Spare
      SPARE3 { ExternalAccessible := 'False'; ExternalVisible := 'False'; ExternalWritable := 'False'} : DWord;   // Spare
      XRAY_KV_DEMAND_ACT { ExternalAccessible := 'False'; ExternalVisible := 'False'; ExternalWritable := 'False'} : Byte;   // X-ray kV demand actual. U8. Expected range 0 to 40kV
      XRAY_MA_DEMAND_ACT { ExternalAccessible := 'False'; ExternalVisible := 'False'; ExternalWritable := 'False'} : Byte;   // X-ray mA demand actual. U8. Expected range 0 to 23mA
      CCYCLE_REP_ACT { ExternalAccessible := 'False'; ExternalVisible := 'False'; ExternalWritable := 'False'} : Byte;   // Checker Cycle repetitions actual. U8. Expected range 0 to 50%
      CALIBRATION_DEV_ACT { ExternalAccessible := 'False'; ExternalVisible := 'False'; ExternalWritable := 'False'} : Byte;   // Calibration deviation actual. U8. Expected range 0 to 8
      EJE_RATE_WARN_LVL_ACT { ExternalAccessible := 'False'; ExternalVisible := 'False'; ExternalWritable := 'False'} : Byte;   // Ejector rate warning level actual. U8. Expected range 0 to 20Ej/sec
      EJE_RATE_ALM_LVL_ACT { ExternalAccessible := 'False'; ExternalVisible := 'False'; ExternalWritable := 'False'} : Byte;   // Ejector rate alarm level actual. U8. Expected range 0 to 20Ej/sec
      BLUE_CALIB_REF_ACT { ExternalAccessible := 'False'; ExternalVisible := 'False'; ExternalWritable := 'False'} : Word;   // Blue calibration reference actual. U16.Expected range 0 to 0 to 10000mV
      RED_CALIB_REF_ACT { ExternalAccessible := 'False'; ExternalVisible := 'False'; ExternalWritable := 'False'} : Word;   // Red calibration reference actual. U16.Expected range 0 to 0 to 10000mV
      PROC_WAT_FLOW_ALM_SP_ACT { ExternalAccessible := 'False'; ExternalVisible := 'False'; ExternalWritable := 'False'} : Byte;   // Process water flow alarm setpoint actual. U8. Expected range 0 to 40litres/min
      PROC_WAT_FLOW_ALM_LVL_DEV_ACT { ExternalAccessible := 'False'; ExternalVisible := 'False'; ExternalWritable := 'False'} : Byte;   // Process water flow alarm level deviation actual. U8. Expected range 0 to 10litres/min
      OVERRIDE_AUD_ALM_ACT { ExternalAccessible := 'False'; ExternalVisible := 'False'; ExternalWritable := 'False'} : Bool;   // Override Audible Alarm Actual - Updated only on Change. ‘0’ – Not overridden, ‘1’ – Overridden
      OVERRIDE_EJE_ALM_ACT { ExternalAccessible := 'False'; ExternalVisible := 'False'; ExternalWritable := 'False'} : Bool;   // Override Ejector Sense Feedback Alarms Actual - Updated only on Change. ‘0’ – Not overridden, ‘1’ – Overridden
      OVERRIDE_CCYCLE_SEQ_ACT { ExternalAccessible := 'False'; ExternalVisible := 'False'; ExternalWritable := 'False'} : Bool;   // Override Checker Cycle Sequence Actual - Updated only on Change. ‘0’ – Not overridden, ‘1’ – Overridden
      MACHINE_TYPE_ACT { ExternalAccessible := 'False'; ExternalVisible := 'False'; ExternalWritable := 'False'} : Bool;   // Machine Type Configured on the cRIO Actual - 1 = Dry 0 = Wet
      DETECTION_TYPE_ACT { ExternalAccessible := 'False'; ExternalVisible := 'False'; ExternalWritable := 'False'} : Bool;   // Machine Detection Type Configured on cRIO Actual - 1 = Dual 0 = Single
      FILM_WINDER_ACT { ExternalAccessible := 'False'; ExternalVisible := 'False'; ExternalWritable := 'False'} : Bool;   // Film Winder Actual. Dry machine only. '0' - Machine has no film winder, '1' - Machine has a film winder.
      SPARE4 { ExternalAccessible := 'False'; ExternalVisible := 'False'; ExternalWritable := 'False'} : Bool;   // Spare
      SPARE5 { ExternalAccessible := 'False'; ExternalVisible := 'False'; ExternalWritable := 'False'} : Bool;   // Spare
      CALIB_DEV_ALM_ENBL_CNT { ExternalAccessible := 'False'; ExternalVisible := 'False'; ExternalWritable := 'False'} : Byte;   // Calibration deviation alarm enable count. U8. Expected range 0 to 8
      SIZEBLU_PMTSETP_ACT_ARR { ExternalAccessible := 'False'; ExternalVisible := 'False'; ExternalWritable := 'False'} : DWord;   // Size of Blue PMT HV set-point actual array. U32. Expect value of 8 elements in array
      BLUPMT_HVSETP_ACT { ExternalAccessible := 'False'; ExternalVisible := 'False'; ExternalWritable := 'False'} : Array[0..7] of Word;   // Blue PMT HV set-point actual. U16[8]. 8 x WORD corresponding to PMT1…PMT8. Expected range 0 to 1200V
      SIZERED_PMTSETP_ACT_ARR { ExternalAccessible := 'False'; ExternalVisible := 'False'; ExternalWritable := 'False'} : DWord;   // Size of Red PMT HV set-point actual array. U32. Expect value of 8 elements in array
      REDPMT_HVSETP_ACT { ExternalAccessible := 'False'; ExternalVisible := 'False'; ExternalWritable := 'False'} : Array[0..7] of Word;   // Red PMT HV set-point actual. U16[8]. 8 x WORD corresponding to PMT1…PMT8. Expected range 0 to 1200V
      SIZEBLU_PMTFDBK_ACT_ARR { ExternalAccessible := 'False'; ExternalVisible := 'False'; ExternalWritable := 'False'} : DWord;   // Size of Blue PMT feedback multiplier actual array. U32. Expect value of 8 elements in array
      BLUPMT_HVFDBK_ACT { ExternalAccessible := 'False'; ExternalVisible := 'False'; ExternalWritable := 'False'} : Array[0..7] of Byte;   // Holds the multiplier value for each blue channel PMT feedback signal: 0 – X1, 1 – X2, 2 – X10, 3 – X50.
      SIZERED_PMTFDBK_ACT_ARR { ExternalAccessible := 'False'; ExternalVisible := 'False'; ExternalWritable := 'False'} : DWord;   // Size of Blue PMT feedback multiplier actual array. U32. Expect value of 8 elements in array
      REDPMT_HVFDBK_ACT { ExternalAccessible := 'False'; ExternalVisible := 'False'; ExternalWritable := 'False'} : Array[0..7] of Byte;   // Holds the multiplier value for each red channel PMT feedback signal: 0 – X1, 1 – X2, 2 – X10, 3 – X50.
      SPARE6 { ExternalAccessible := 'False'; ExternalVisible := 'False'; ExternalWritable := 'False'} : DWord;   // Spare
      SPARE7 { ExternalAccessible := 'False'; ExternalVisible := 'False'; ExternalWritable := 'False'} : DWord;   // Spare
      SPARE8 { ExternalAccessible := 'False'; ExternalVisible := 'False'; ExternalWritable := 'False'} : DWord;   // Spare
      SPARE9 { ExternalAccessible := 'False'; ExternalVisible := 'False'; ExternalWritable := 'False'} : DWord;   // Spare
      SPARE10 { ExternalAccessible := 'False'; ExternalVisible := 'False'; ExternalWritable := 'False'} : DWord;   // Spare
      SPARE11 { ExternalAccessible := 'False'; ExternalVisible := 'False'; ExternalWritable := 'False'} : Word;   // Spare
      COOLWAT_FLOW_RATE { ExternalAccessible := 'False'; ExternalVisible := 'False'; ExternalWritable := 'False'} : Byte;   // Cooling water flow rate. U8. Sensor feedback. Expected range 0 to 20 litres/min.
      COOLWAT_TEMP { ExternalAccessible := 'False'; ExternalVisible := 'False'; ExternalWritable := 'False'} : Byte;   // Cooling water temperature. U8. Sensor feedback. Expected range 0 to 100⁰C.
      INCOM_AIR_PRESS { ExternalAccessible := 'False'; ExternalVisible := 'False'; ExternalWritable := 'False'} : Word;   // Incoming air pressure. U16. Sensor feedback. Expected range 0 to 1000 which equates to 0 to 10.00bar.
      PROCWAT_FLOW_RATE { ExternalAccessible := 'False'; ExternalVisible := 'False'; ExternalWritable := 'False'} : Word;   // Process water flow rate. U16. Sensor feedback. Expected range 0 to 4500 which equates to 0 to 45.00 litres/min. (Wet machine only)
      XRAY_GEN_COMP_TEMP { ExternalAccessible := 'False'; ExternalVisible := 'False'; ExternalWritable := 'False'} : Byte;   // X-ray generator compartment temperature. U8. Sensor feedback. Expected range 0 to 100⁰C.
      XRAY_KV_FEEDBK { ExternalAccessible := 'False'; ExternalVisible := 'False'; ExternalWritable := 'False'} : Byte;   // X-ray kV feedback. U8. X-ray feedback. Expected range 0 to 60kV.
      XRAY_MA_FEEDBK { ExternalAccessible := 'False'; ExternalVisible := 'False'; ExternalWritable := 'False'} : Byte;   // X-ray mA feedback. U8. X-ray feedback. Expected range 0 to 25mA.
      HEARTBEAT_CRIOCONT_MPLC { ExternalAccessible := 'False'; ExternalVisible := 'False'; ExternalWritable := 'False'} : Byte;   // Communications heartbeat from CRIO Controller to Machine PLC. Returns value received in PLC control message.
      LOOKUP_TABLE_USER_NAME { ExternalAccessible := 'False'; ExternalVisible := 'False'; ExternalWritable := 'False'} : Array[0..7] of Byte;   // Lookup table username. Username at requested security lookup table pointer, 8-character string
      LOOKUP_TABLE_ACCESS_LVL { ExternalAccessible := 'False'; ExternalVisible := 'False'; ExternalWritable := 'False'} : Byte;   // Lookup table access level. Access level at requested security lookup table pointer
      LOGGED_ON_USER_ACCES_LVL { ExternalAccessible := 'False'; ExternalVisible := 'False'; ExternalWritable := 'False'} : Byte;   // Access level for the current logged on user: 0-Operator (default)1-Technician2-Metallurgist 3-Administrator
      CURRENT_USER_NAME { ExternalAccessible := 'False'; ExternalVisible := 'False'; ExternalWritable := 'False'} : Array[0..7] of Byte;   // Current User Name Logged On to the cRIO, 8 character string
      VIB_FEED_FEEDBK { ExternalAccessible := 'False'; ExternalVisible := 'False'; ExternalWritable := 'False'} : Byte;   // Vibratory feeder feedback. U8. Feeder feedback. Expected range 0 to 100% full scale deflection.
      GATE_POS_ACT { ExternalAccessible := 'False'; ExternalVisible := 'False'; ExternalWritable := 'False'} : Byte;   // Reflects the current/actual position of the Auto gate if present. ‘0’ - No auto gate, '1’ – gate at position1(-2 +1mm), '2’ – gate at position2(-4 +2mm), '3’ – Gate at position3(-8 +4mm), '4’ – Gate at position4(-16 +8mm), '5’ – Gate at position5(-32 +16mm)
      REMOTE_REC_TO_UPDATE { ExternalAccessible := 'False'; ExternalVisible := 'False'; ExternalWritable := 'False'} : Byte;   // 1 x BYTE corresponding to 0-15, 0 = no action, 1-15 = copy current recipe values to this recipe destination e.g. 5 = copy current recipe values to remote recipe 5.
      CRIO_CONT_TIME_HRS { ExternalAccessible := 'False'; ExternalVisible := 'False'; ExternalWritable := 'False'} : Byte;   // System time - hours: 0 - 23
      CRIO_CONT_TIME_MINS { ExternalAccessible := 'False'; ExternalVisible := 'False'; ExternalWritable := 'False'} : Byte;   // System time - minutes: 0 - 59
      CRIO_CONT_TIME_SECS { ExternalAccessible := 'False'; ExternalVisible := 'False'; ExternalWritable := 'False'} : Byte;   // System time - seconds: 0 - 59
      CRIO_CONT_TIME_CEN { ExternalAccessible := 'False'; ExternalVisible := 'False'; ExternalWritable := 'False'} : Byte;   // System date - centuary : 0 - 99
      CRIO_CONT_TIME_YRS { ExternalAccessible := 'False'; ExternalVisible := 'False'; ExternalWritable := 'False'} : Byte;   // System date - year: 0 - 99
      CRIO_CONT_TIME_MNT { ExternalAccessible := 'False'; ExternalVisible := 'False'; ExternalWritable := 'False'} : Byte;   // System date - month: 1-12
      CRIO_CONT_TIME_DAY { ExternalAccessible := 'False'; ExternalVisible := 'False'; ExternalWritable := 'False'} : Byte;   // System date - day: 1-31
      MACH_POWER_CONSUMP { ExternalAccessible := 'False'; ExternalVisible := 'False'; ExternalWritable := 'False'} : DWord;   // U32. Running total of power consumption in kWh of the machine.
      MACH_PROCWATER_CONSUMP { ExternalAccessible := 'False'; ExternalVisible := 'False'; ExternalWritable := 'False'} : DWord;   // U32. Running total process water consumption in kilo litres of the machine.
      FEEDER_STOPPED_STATUS { ExternalAccessible := 'False'; ExternalVisible := 'False'; ExternalWritable := 'False'} : Byte;   // Reason why feeder is not running in Processing state or feeder cannot be started in Processing Ready state.Reason why feeder is not running in Processing state or feeder cannot be started in Processing Ready state. 0 – none (feeder is running or can be started); 1 – Processing water flow low; 2 – Incoming air pressure low low; 3 – Ejection rate alarm; 4 – Downstream interlock
      SPARE12 { ExternalAccessible := 'False'; ExternalVisible := 'False'; ExternalWritable := 'False'} : Byte;   // Spare
      SPARE13 { ExternalAccessible := 'False'; ExternalVisible := 'False'; ExternalWritable := 'False'} : DWord;   // Spare
      SPARE14 { ExternalAccessible := 'False'; ExternalVisible := 'False'; ExternalWritable := 'False'} : DWord;   // Spare
      SPARE15 { ExternalAccessible := 'False'; ExternalVisible := 'False'; ExternalWritable := 'False'} : DWord;   // Spare
      BLUE_PEAK_INTEN { ExternalAccessible := 'False'; ExternalVisible := 'False'; ExternalWritable := 'False'} : Word;   // Blue Peak Intensity. U16. Holds blue value of last detection. Expected range 0 to 10000mV
      RED_PEAK_INTEN { ExternalAccessible := 'False'; ExternalVisible := 'False'; ExternalWritable := 'False'} : Word;   // Red Peak Intensity. U16. Holds red value of last peak detection. Expected range 0 to 10000mV
      MOST_ACTIVE_FIRE_CHAN { ExternalAccessible := 'False'; ExternalVisible := 'False'; ExternalWritable := 'False'} : Byte;   // Most active fire rate channel. U8. Indicates the channel that currently has the highest firing rate. Expected range 0 to 8
      MOST_ACTIVE_CHAN_FIRE { ExternalAccessible := 'False'; ExternalVisible := 'False'; ExternalWritable := 'False'} : Byte;   // Most active channel firing rate. U8. Indicates the most active channels firing rate [ej/sec] multiplied by 10 i.e. 225 received therefore indicates 22.5 ej/sec
      LAST_EJECT_ACTIV { ExternalAccessible := 'False'; ExternalVisible := 'False'; ExternalWritable := 'False'} : Byte;   // Last Ejector Activated. Indicates the channel of the last ejector activated. Expected range 0 to 8
      SPARE16 { ExternalAccessible := 'False'; ExternalVisible := 'False'; ExternalWritable := 'False'} : Byte;   // Spare
      RES_NUMELEM_IN_ARRAY_0 { ExternalAccessible := 'False'; ExternalVisible := 'False'; ExternalWritable := 'False'} : DWord;   // Reserved (Holds number of elements in array)
      EJECT_DELAY_RESP { ExternalAccessible := 'False'; ExternalVisible := 'False'; ExternalWritable := 'False'} : Array[0..15] of Byte;   // 16 x BYTE corresponding to CH1_1…CH8_2. Expected range 0 to 255
      RES_NUMELEM_IN_ARRAY_1 { ExternalAccessible := 'False'; ExternalVisible := 'False'; ExternalWritable := 'False'} : DWord;   // Reserved (Holds number of elements in array)
      EJECT_DUR_RESP { ExternalAccessible := 'False'; ExternalVisible := 'False'; ExternalWritable := 'False'} : Array[0..15] of Byte;   // 16 x BYTE corresponding to CH1_1…CH8_2. Expected range 0 to 255
      RES_NUMELEM_IN_ARRAY_2 { ExternalAccessible := 'False'; ExternalVisible := 'False'; ExternalWritable := 'False'} : DWord;   // Reserved (Holds number of elements in array)
      EJECT_ERROR_HIST { ExternalAccessible := 'False'; ExternalVisible := 'False'; ExternalWritable := 'False'} : Array[0..15] of DWord;   // 16 x DWORD corresponding to CH1_1…CH8_2 (64 bytes)
      RES_NUMELEM_IN_ARRAY_3 { ExternalAccessible := 'False'; ExternalVisible := 'False'; ExternalWritable := 'False'} : DWord;   // Reserved (Holds number of elements in array)
      EJECT_PROFILE { ExternalAccessible := 'False'; ExternalVisible := 'False'; ExternalWritable := 'False'} : Array[0..7] of DWord;   // 8 x DWORD corresponding to CH1…CH8 (32 bytes)
      RES_NUMELEM_IN_ARRAY_4 { ExternalAccessible := 'False'; ExternalVisible := 'False'; ExternalWritable := 'False'} : DWord;   // Reserved (Holds number of elements in array)
      ACCEP_PROFILE { ExternalAccessible := 'False'; ExternalVisible := 'False'; ExternalWritable := 'False'} : Array[0..7] of DWord;   // 8 x DWORD corresponding to CH1…CH8 (32 bytes)
      RES_NUMELEM_IN_ARRAY_5 { ExternalAccessible := 'False'; ExternalVisible := 'False'; ExternalWritable := 'False'} : DWord;   // Reserved (Holds number of elements in array)
      REJECT_PROFILE { ExternalAccessible := 'False'; ExternalVisible := 'False'; ExternalWritable := 'False'} : Array[0..7] of DWord;   // 8 x DWORD corresponding to CH1…CH8 (32 bytes)
      RES_NUMELEM_IN_ARRAY_6 { ExternalAccessible := 'False'; ExternalVisible := 'False'; ExternalWritable := 'False'} : DWord;   // Reserved (Holds number of elements in array)
      BLUE_CALIB_REF_DATA { ExternalAccessible := 'False'; ExternalVisible := 'False'; ExternalWritable := 'False'} : Array[0..7] of Word;   // 8 x WORD corresponding to CH1…CH8 (16 bytes)
      RES_NUMELEM_IN_ARRAY_7 { ExternalAccessible := 'False'; ExternalVisible := 'False'; ExternalWritable := 'False'} : DWord;   // Reserved (Holds number of elements in array)
      BLUE_CALIB_CC_DATA { ExternalAccessible := 'False'; ExternalVisible := 'False'; ExternalWritable := 'False'} : Array[0..7] of Word;   // 8 x WORD corresponding to CH1…CH8 (16 bytes)
      RES_NUMELEM_IN_ARRAY_8 { ExternalAccessible := 'False'; ExternalVisible := 'False'; ExternalWritable := 'False'} : DWord;   // Reserved (Holds number of elements in array)
      RED_CALIB_REF_DATA { ExternalAccessible := 'False'; ExternalVisible := 'False'; ExternalWritable := 'False'} : Array[0..7] of Word;   // 8 x WORD corresponding to CH1…CH8 (16 bytes)
      RES_NUMELEM_IN_ARRAY_9 { ExternalAccessible := 'False'; ExternalVisible := 'False'; ExternalWritable := 'False'} : DWord;   // Reserved (Holds number of elements in array)
      RED_CALIB_CC_DATA { ExternalAccessible := 'False'; ExternalVisible := 'False'; ExternalWritable := 'False'} : Array[0..7] of Word;   // 8 x WORD corresponding to CH1…CH8 (16 bytes)
      RES_NUMELEM_IN_ARRAY_10 { ExternalAccessible := 'False'; ExternalVisible := 'False'; ExternalWritable := 'False'} : DWord;   // Reserved (Holds number of elements in array)
      ACCEPT_LI_HIST { ExternalAccessible := 'False'; ExternalVisible := 'False'; ExternalWritable := 'False'} : Array[0..63] of DWord;   // 64 x DWORD corresponding to bin no 1…64 (256 bytes)
      RES_NUMELEM_IN_ARRAY_11 { ExternalAccessible := 'False'; ExternalVisible := 'False'; ExternalWritable := 'False'} : DWord;   // Reserved (Holds number of elements in array)
      REJECT_LI_HIST { ExternalAccessible := 'False'; ExternalVisible := 'False'; ExternalWritable := 'False'} : Array[0..63] of DWord;   // 64 x DWORD corresponding to bin no 1…64 (256 bytes)
      RES_NUMELEM_IN_ARRAY_12 { ExternalAccessible := 'False'; ExternalVisible := 'False'; ExternalWritable := 'False'} : DWord;   // Reserved (Holds number of elements in array)
      RED_LI_HIST { ExternalAccessible := 'False'; ExternalVisible := 'False'; ExternalWritable := 'False'} : Array[0..63] of DWord;   // 64 x DWORD corresponding to bin no 1…64 (256 bytes)
      RES_NUMELEM_IN_ARRAY_13 { ExternalAccessible := 'False'; ExternalVisible := 'False'; ExternalWritable := 'False'} : DWord;   // Reserved (Holds number of elements in array)
      BLUE_RED_RATIO_LI_HIST { ExternalAccessible := 'False'; ExternalVisible := 'False'; ExternalWritable := 'False'} : Array[0..63] of DWord;   // 64 x DWORD corresponding to bin no 1…64 (256 bytes)
      LI_HIST_CLR_TIME_HRS { ExternalAccessible := 'False'; ExternalVisible := 'False'; ExternalWritable := 'False'} : Byte;   // LI histogram clear time - hours: 0 - 23
      LI_HIST_CLR_TIME_MINS { ExternalAccessible := 'False'; ExternalVisible := 'False'; ExternalWritable := 'False'} : Byte;   // LI histogram clear time - minutes: 0 - 59
      LI_HIST_CLR_TIME_SECS { ExternalAccessible := 'False'; ExternalVisible := 'False'; ExternalWritable := 'False'} : Byte;   // LI histogram clear time - seconds: 0 - 59
      LI_HIST_CLR_DATE_CENT { ExternalAccessible := 'False'; ExternalVisible := 'False'; ExternalWritable := 'False'} : Byte;   // LI histogram clear date - centuary : 0 - 99
      LI_HIST_CLR_DATE_YRS { ExternalAccessible := 'False'; ExternalVisible := 'False'; ExternalWritable := 'False'} : Byte;   // LI histogram clear date - year: 0 - 99
      LI_HIST_CLR_DATE_MNT { ExternalAccessible := 'False'; ExternalVisible := 'False'; ExternalWritable := 'False'} : Byte;   // LI histogram clear date - month: 1-12
      LI_HIST_CLR_DATE_DAY { ExternalAccessible := 'False'; ExternalVisible := 'False'; ExternalWritable := 'False'} : Byte;   // LI histogram clear date - day: 1-31
      SPARE17 { ExternalAccessible := 'False'; ExternalVisible := 'False'; ExternalWritable := 'False'} : Byte;   // Spare
      TIME_SINCE_HIST_CLR { ExternalAccessible := 'False'; ExternalVisible := 'False'; ExternalWritable := 'False'} : DWord;   // DWORD indicating the time difference between the Current Time and the Histogram Clear Time, in seconds
      SPARE18 { ExternalAccessible := 'False'; ExternalVisible := 'False'; ExternalWritable := 'False'} : DWord;   // Spare
      SPARE19 { ExternalAccessible := 'False'; ExternalVisible := 'False'; ExternalWritable := 'False'} : DWord;   // Spare
      SPARE20 { ExternalAccessible := 'False'; ExternalVisible := 'False'; ExternalWritable := 'False'} : DWord;   // Spare
      SPARE21 { ExternalAccessible := 'False'; ExternalVisible := 'False'; ExternalWritable := 'False'} : DWord;   // Spare
      SPARE22 { ExternalAccessible := 'False'; ExternalVisible := 'False'; ExternalWritable := 'False'} : DWord;   // Spare
      SPARE23 { ExternalAccessible := 'False'; ExternalVisible := 'False'; ExternalWritable := 'False'} : DWord;   // Spare
   END_STRUCT;
END_TYPE
